(* IEC 61131-3 sources: plcc/tests/fixtures/parse, 10 files *)

(* ---- pou_function.st ---- *)
FUNCTION ABS_INT : INT
VAR_INPUT
    value : INT;
END_VAR
    IF value < 0 THEN
        ABS_INT := -value;
    ELSE
        ABS_INT := value;
    END_IF;
END_FUNCTION

FUNCTION Clamp : REAL
VAR_INPUT
    value : REAL;
    low : REAL;
    high : REAL;
END_VAR
    IF value < low THEN
        Clamp := low;
    ELSIF value > high THEN
        Clamp := high;
    ELSE
        Clamp := value;
    END_IF;
END_FUNCTION

(* ---- oop.st ---- *)
INTERFACE IMovable
    METHOD Move : BOOL
    VAR_INPUT
        dx : REAL;
        dy : REAL;
    END_VAR
    END_METHOD
END_INTERFACE

CLASS Shape IMPLEMENTS IMovable
VAR
    pos_x : REAL := 0.0;
    pos_y : REAL := 0.0;
END_VAR
    METHOD Move : BOOL
    VAR_INPUT
        dx : REAL;
        dy : REAL;
    END_VAR
        pos_x := pos_x + dx;
        pos_y := pos_y + dy;
        Move := TRUE;
    END_METHOD

    METHOD GetX : REAL
        GetX := pos_x;
    END_METHOD

    METHOD GetY : REAL
        GetY := pos_y;
    END_METHOD
END_CLASS

FUNCTION_BLOCK Circle EXTENDS Shape
VAR
    radius : REAL := 1.0;
END_VAR
    METHOD Area : REAL
        Area := 3.14159 * radius * radius;
    END_METHOD
END_FUNCTION_BLOCK

(* ---- pou_function_block.st ---- *)
FUNCTION_BLOCK TON_Simple
VAR_INPUT
    IN_SIGNAL : BOOL;
    PT : INT;
END_VAR
VAR_OUTPUT
    Q : BOOL;
    ET : INT;
END_VAR
VAR
    running : BOOL := FALSE;
    elapsed : INT := 0;
END_VAR
    IF IN_SIGNAL THEN
        IF NOT running THEN
            running := TRUE;
            elapsed := 0;
        END_IF;
        IF running AND NOT Q THEN
            elapsed := elapsed + 1;
            IF elapsed >= PT THEN
                Q := TRUE;
                ET := PT;
            ELSE
                ET := elapsed;
            END_IF;
        END_IF;
    ELSE
        running := FALSE;
        Q := FALSE;
        ET := 0;
        elapsed := 0;
    END_IF;
END_FUNCTION_BLOCK

(* ---- variables.st ---- *)
FUNCTION_BLOCK VarTest
VAR_INPUT
    in1 : INT;
    in2 : BOOL;
END_VAR
VAR_OUTPUT
    out1 : INT;
    out2 : REAL;
END_VAR
VAR_IN_OUT
    inout1 : INT;
END_VAR
VAR
    local1 : INT := 0;
    local2 : REAL := 1.0;
END_VAR
VAR_TEMP
    temp1 : INT;
END_VAR
VAR CONSTANT
    PI : REAL := 3.14159;
    MAX_COUNT : INT := 1000;
END_VAR
VAR RETAIN
    persistent_counter : INT := 0;
END_VAR
    out1 := in1 + local1;
END_FUNCTION_BLOCK

(* ---- direct_representation.st ---- *)
PROGRAM DirectRep
VAR
    input_word AT %IW0 : WORD;
    output_byte AT %QB0 : BYTE;
    memory_bit AT %MX0.0 : BOOL;
    memory_dword AT %MD10 : DWORD;
END_VAR
    output_byte := 16#FF;
    memory_bit := TRUE;
END_PROGRAM

(* ---- expressions.st ---- *)
PROGRAM TestExpressions
VAR
    a : INT := 0;
    b : INT := 0;
    c : INT := 0;
    d : REAL := 0.0;
    flag : BOOL := FALSE;
END_VAR
    (* Arithmetic *)
    a := 1 + 2;
    a := 3 - 1;
    a := 2 * 3;
    a := 10 / 2;
    a := 10 MOD 3;
    d := 2.0 ** 3.0;

    (* Comparison *)
    flag := a = b;
    flag := a <> b;
    flag := a < b;
    flag := a <= b;
    flag := a > b;
    flag := a >= b;

    (* Logical *)
    flag := TRUE AND FALSE;
    flag := TRUE OR FALSE;
    flag := TRUE XOR FALSE;
    flag := NOT flag;
    flag := TRUE & FALSE;

    (* Precedence *)
    a := 1 + 2 * 3;
    a := (1 + 2) * 3;

    (* Nested *)
    a := (a + b) * (c - 1);
END_PROGRAM

(* ---- literals.st ---- *)
PROGRAM TestLiterals
VAR
    b : BOOL := TRUE;
    i : INT := 42;
    hex : DINT := 16#FF;
    bin : BYTE := 2#10101010;
    oct : INT := 8#77;
    r : REAL := 3.14;
    s : STRING := 'Hello, World!';
    neg : INT := -1;
    big : LINT := 1_000_000;
    typed_int : INT := INT#100;
    typed_real : REAL := REAL#2.718;
    typed_bool : BOOL := BOOL#TRUE;
END_VAR
END_PROGRAM

(* ---- pou_program.st ---- *)
PROGRAM MultiVarBlocks
VAR_INPUT
    start_cmd : BOOL;
    stop_cmd : BOOL;
END_VAR
VAR_OUTPUT
    running : BOOL;
    error : BOOL;
END_VAR
VAR
    state : INT := 0;
    cycle_count : DINT := 0;
END_VAR
    IF stop_cmd THEN
        running := FALSE;
        state := 0;
    ELSIF start_cmd THEN
        running := TRUE;
        state := 1;
    END_IF;

    IF running THEN
        cycle_count := cycle_count + 1;
    END_IF;
END_PROGRAM

(* ---- statements.st ---- *)
PROGRAM TestStatements
VAR
    x : INT := 0;
    y : INT := 0;
    flag : BOOL := FALSE;
    sum : INT := 0;
    i : INT;
END_VAR
    (* Assignment *)
    x := 42;

    (* IF / ELSIF / ELSE *)
    IF x > 10 THEN
        y := 1;
    ELSIF x > 5 THEN
        y := 2;
    ELSIF x > 0 THEN
        y := 3;
    ELSE
        y := 0;
    END_IF;

    (* CASE *)
    CASE x OF
        0:
            flag := FALSE;
        1, 2, 3:
            flag := TRUE;
        10..20:
            y := 100;
    ELSE
        y := -1;
    END_CASE;

    (* FOR *)
    sum := 0;
    FOR i := 1 TO 100 BY 2 DO
        sum := sum + i;
    END_FOR;

    (* WHILE *)
    WHILE sum > 0 DO
        sum := sum - 1;
    END_WHILE;

    (* REPEAT..UNTIL *)
    REPEAT
        sum := sum + 1;
    UNTIL sum >= 50
    END_REPEAT;

    (* EXIT / CONTINUE *)
    FOR i := 0 TO 100 DO
        IF i = 50 THEN
            EXIT;
        END_IF;
        IF i MOD 2 = 0 THEN
            CONTINUE;
        END_IF;
        sum := sum + i;
    END_FOR;

    (* RETURN *)
    RETURN;
END_PROGRAM

(* ---- types.st ---- *)
TYPE
    Color : (Red, Green, Blue);
END_TYPE

TYPE
    Voltage : REAL;
END_TYPE

TYPE
    SmallInt : INT(0..100);
END_TYPE

TYPE
    TenInts : ARRAY[0..9] OF INT;
END_TYPE

TYPE
    Point : STRUCT
        x : REAL := 0.0;
        y : REAL := 0.0;
        z : REAL := 0.0;
    END_STRUCT;
END_TYPE

PROGRAM TypesTest
VAR
    color : Color := Color#Red;
    volts : Voltage := 3.3;
    small : SmallInt := 50;
    arr : TenInts;
    pt : Point;
    matrix : ARRAY[0..2, 0..2] OF REAL;
    name : STRING[80] := 'test';
END_VAR
    arr[0] := 42;
    pt.x := 1.0;
    pt.y := 2.0;
    matrix[0, 0] := 1.0;
END_PROGRAM
